//{attribute 'qualified_only'}
VAR_GLOBAL
	GVL_DUT_TC_AP240ACPower					: DUT_Cylinder;
	GVL_DUT_DC_AP240ACPower					: DUT_Cylinder;
END_VAR

(* stored: Version 1.1.0.1, ProductVersion 3.1.4022.18
   GVL GVL_Motor: Id {8ded2be3-72f2-4213-9223-57e7e250d32d} *)
